// TIA Portal V20 export
DATA_BLOCK "DB_CommPLC_ISO"   // DB1100
// stored: AutoNumber false, InstanceOfName FB_CommPLC_ISO, InstanceOfType FB
"FB_CommPLC_ISO"
   // VAR
   //    sSynchro_ULx { ExternalVisible := 'False'; ExternalWritable := 'False'} : Byte;
   //    sSynchro_ULx_WriteON { ExternalAccessible := 'False'; ExternalVisible := 'False'; ExternalWritable := 'False'} : Bool;
   //    sRT_FixtureVW_Rel : R_TRIG;
   //    sRT_FixtureVW_Req { S7_SetPoint := 'True'} : R_TRIG;
   //    sRT_GripperAvail { S7_SetPoint := 'True'} : R_TRIG;
   //    sAxisManagedByNC { S7_SetPoint := 'True'} : Bool;
   //    sAxisReservedbyNC : Bool;
   // END_VAR
BEGIN
END_DATA_BLOCK
